TYPE ST_HMI_Page :
STRUCT
	Home_page		: BOOL;
	Allarms_page	: BOOL;
	Params_page		: BOOL;
	
	Numbers_page	: INT;	//0	Home
							//1 Allarms
							//2 Params
	
END_STRUCT
END_TYPE

(* stored: Version 1.1.0.1, ProductVersion 3.1.4024.12
   DUT ST_HMI_Page: Id {f7a7f018-6f3d-404c-8f7e-da5ba158cdd1} *)
